// TIA Portal V20 export
DATA_BLOCK "SBK09"   // DB209
// stored: MemoryReserve 100
   VAR
      "X1-0 Gate ScrapBox: Lock" : Bool;
      "X2-1 Gate ScrapBox : Reset" : Bool;
      "X3-2 reserved" : Bool;
      "X4-3 reserved" : Bool;
      "X1-4 Gate ScrapBox : Unlock" : Bool;
      "X2-5 reserved" : Bool;
      "X3-6 reserved" : Bool;
      "X4-7 reserved" : Bool;
      "X5-0 Gate ScrapBox : Lock lamp on" : Bool;
      "X6-1 Gate ScrapBox : Unlock lamp on" : Bool;
      "X7-2 Gate ScrapBox : Reset lamp on" : Bool;
   END_VAR
BEGIN
END_DATA_BLOCK
